// TIA Portal V20 export
FUNCTION "Drivers_To_Move_Pallet" : Void   // FC5, LAD
{ S7_Optimized_Access := 'TRUE' }
// stored: SetENOAutomatically false
   VAR_INPUT
      HW_Driver : HW_IO;
      Reset : Bool;
   END_VAR
   VAR_IN_OUT
      iDrive_Param : "SEW_MOVIKIT_VelocityDrive_SETPOINTS_V2.1";
      oDrive_Param : "SEW_MOVIKIT_VelocityDrive_STATUS_V2.1";
   END_VAR
   VAR_TEMP
      Communication_OK : Bool;
   END_VAR
BEGIN

REGION Network 1
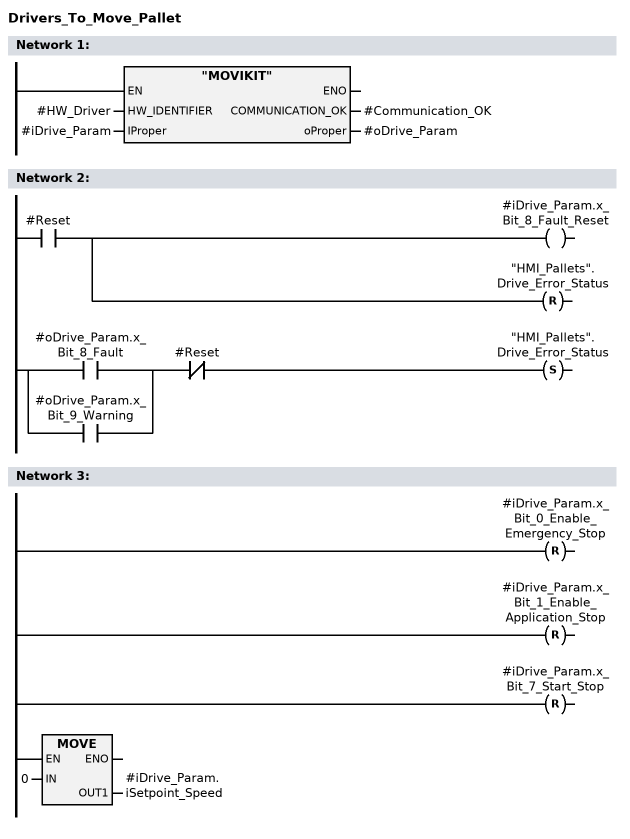
   RUNG wire#powerrail
      "MOVIKIT"(HW_IDENTIFIER := #HW_Driver, IProper := #iDrive_Param, COMMUNICATION_OK => #Communication_OK, oProper => #oDrive_Param)
   END_RUNG
   // the same network as SCL:
   "MOVIKIT"(HW_IDENTIFIER := #HW_Driver,
             IProper := #iDrive_Param,
             COMMUNICATION_OK => #Communication_OK,
             oProper => #oDrive_Param);
END_REGION

REGION Network 2
   RUNG wire#powerrail
      Contact( #Reset )
      wire#w1
      Coil( #iDrive_Param.x_Bit_8_Fault_Reset )
   END_RUNG
   RUNG wire#w1
      R_Coil( "HMI_Pallets".Drive_Error_Status )
   END_RUNG
   RUNG wire#powerrail
      Contact( #oDrive_Param.x_Bit_8_Fault )
      wire#w2
      I_Contact( #Reset )
      S_Coil( "HMI_Pallets".Drive_Error_Status )
   END_RUNG
   RUNG wire#powerrail
      Contact( #oDrive_Param.x_Bit_9_Warning )
   END_RUNG wire#w2
   // the same network as SCL:
   #iDrive_Param.x_Bit_8_Fault_Reset := #Reset;
   IF #Reset THEN "HMI_Pallets".Drive_Error_Status := FALSE; END_IF;
   IF (#oDrive_Param.x_Bit_8_Fault OR #oDrive_Param.x_Bit_9_Warning) AND NOT #Reset THEN
       "HMI_Pallets".Drive_Error_Status := TRUE;
   END_IF;
END_REGION

REGION Network 3
   RUNG wire#powerrail
      R_Coil( #iDrive_Param.x_Bit_0_Enable_Emergency_Stop )
   END_RUNG
   RUNG wire#powerrail
      R_Coil( #iDrive_Param.x_Bit_1_Enable_Application_Stop )
   END_RUNG
   RUNG wire#powerrail
      R_Coil( #iDrive_Param.x_Bit_7_Start_Stop )
   END_RUNG
   RUNG wire#powerrail
      Move(in := 0, out1 => #iDrive_Param.iSetpoint_Speed)
   END_RUNG
   // the same network as SCL:
   #iDrive_Param.x_Bit_0_Enable_Emergency_Stop := FALSE;
   #iDrive_Param.x_Bit_1_Enable_Application_Stop := FALSE;
   #iDrive_Param.x_Bit_7_Start_Stop := FALSE;
   #iDrive_Param.iSetpoint_Speed := 0;
END_REGION
END_FUNCTION
